// TIA Portal V16 export
// export: Created 2023-03-29T11:04:42.156007Z, ExportSetting WithDefaults, DisplayName Totally Integrated Automation Portal, DisplayVersion V16 Update 6, DisplayName TIA Portal Version Control Interface, DisplayVersion V16 Update 2, DisplayName TIA Portal Openness, DisplayVersion V16 Update 6, DisplayName STEP 7 Professional, DisplayVersion V16 Update 6, DisplayName STEP 7 Safety, DisplayVersion V16, DisplayName WinCC Advanced, DisplayVersion V16 Update 6
DATA_BLOCK "dbMasterData"   // DB35
{ S7_Optimized_Access := 'FALSE' }
VERSION : 0.1
// stored: AutoNumber false, DBAccessibleFromOPCUA true, IsOnlyStoredInLoadMemory false, IsWriteProtectedInAS false
   VAR
      data5_Wielkość_przeływu_Adres_0 { S7_SetPoint := 'True'} : "typeDataMPP04_Int";   // wielkość przepływu / Wartość aktualnego przepływu
      data5_Licznik_objętość_VF_Adres_2 : "typeDataMPP04_Int";   // licznik objętości VF / Stan licznika objętości dla przepływu w przód VF
      data5_Licznik_objętość_VR_Adres_4 { S7_SetPoint := 'True'} : "typeDataMPP04_Int";   // licznik objętości VR / Stan licznika objętości dla przepływu w tył VR
      data5_Licznik_różnicowy_VD_Adres_6 { S7_SetPoint := 'True'} : "typeDataMPP04_Int";   // licznik różnicy / Stan bieżącego różnicowego licznika objętości VD
      data5_Stan_licz_bjętości_GF_Adres_8 { S7_SetPoint := 'True'} : "typeDataMPP04_Int";   // licznik objetosci GF / Stan głównego licznika objętości dla przepływu w przód GF
      data5_Stan_licz_bjętości_GR_Adres_10 { S7_SetPoint := 'True'} : "typeDataMPP04_Int";   // licznik objetości GR / Sta ngłownego licznika objętości dla przepływu w tył GR
      data5_Stan_licz_rózicowego_obj_GD_Adres_12 { S7_SetPoint := 'True'} : "typeDataMPP04_Int";   // licznik róznicowy / Stan głownego licznika różnicowego GD
      data5_Stan_urządzenia_1000 { S7_SetPoint := 'True'} : "typeDataInverter_Word";   // stan urządzenia / 8-przekrodzony zakres pracy przetwornika, 20-otwarty obwód cewki, 21zwarcie w obwodzie cewki, 26-brak cieczy w czujniku
      data6_Wielkość_przeływu_Adres_0 { S7_SetPoint := 'True'} : "typeDataMPP04_Int";   // wielkość przepływu / Wartość aktualnego przepływu
      data6_Licznik_objętość_VF_Adres_2 { S7_SetPoint := 'True'} : "typeDataMPP04_Int";   // licznik objętości VF / Stan licznika objętości dla przepływu w przód VF
      data6_Licznik_objętość_VR_Adres_4 { S7_SetPoint := 'True'} : "typeDataMPP04_Int";   // licznik objętości VR / Stan licznika objętości dla przepływu w tył VR
      data6_Licznik_różnicowy_VD_Adres_6 { S7_SetPoint := 'True'} : "typeDataMPP04_Int";   // licznik różnicy / Stan bieżącego różnicowego licznika objętości VD
      data6_Stan_licz_bjętości_GF_Adres_8 { S7_SetPoint := 'True'} : "typeDataMPP04_Int";   // licznik objetosci GF / Stan głównego licznika objętości dla przepływu w przód GF
      data6_Stan_licz_bjętości_GR_Adres_10 { S7_SetPoint := 'True'} : "typeDataMPP04_Int";   // licznik objetości GR / Sta ngłownego licznika objętości dla przepływu w tył GR
      data6_Stan_licz_rózicowego_obj_GD_Adres_12 { S7_SetPoint := 'True'} : "typeDataMPP04_Int";   // licznik róznicowy / Stan głownego licznika różnicowego GD
      data6_Stan_urządzenia_1000 { S7_SetPoint := 'True'} : "typeDataInverter_Word";   // stan urządzenia / 8-przekrodzony zakres pracy przetwornika, 20-otwarty obwód cewki, 21zwarcie w obwodzie cewki, 26-brak cieczy w czujniku
      data26_Inver_Control_word_416000_Fal { S7_SetPoint := 'True'} : "typeDataInverter_Word";   // Sowo komtrolneCTW falownika [Uint16, index 0]
      data26_Inver_setpoint_ref_416020_Fal { S7_SetPoint := 'True'} : "typeDataInverter_Word";   // Słowo wartość zadana Hz [Int16, index -1]
      data26_Inver_Status_word_416030_Fal { S7_SetPoint := 'True'} : "typeDataInverter_Word";   // Słowo statusu STW falownika [Uint16, index 0]
      data26_Inver_Frequency_416130_Fal { S7_SetPoint := 'True'} : "typeDataInverter_Word";   // Słowo częstotliwość na wyjściu [Uint16, index -1]
      data26_Inver_MotorCurrent_416140_Fal { S7_SetPoint := 'True'} : "typeDataInverter_Word";   // Słowo częstotliwość na wyjściu [Uint16, index -2]
      data26_Inver_DC_Voltage_416300_Fal { S7_SetPoint := 'True'} : "typeDataInverter_Word";   // Słowo napięcia DC na szynie [Uint16, index 0]
      data26_Inver_Temp_416340_Fal { S7_SetPoint := 'True'} : "typeDataInverter_Word";   // Słowo temperatura invertera [Uint8, index 0]
      data26_Inver_NomCurrent_416360_Fal { S7_SetPoint := 'True'} : "typeDataInverter_Word";   // Słowo nominalna wartośc prądu falonika[Uint16, index -2]
      data26_Inver_MaxCurrent_416370_Fal { S7_SetPoint := 'True'} : "typeDataInverter_Word";   // Słowo max prąd falownika [Uint16, index -2]
      data26_Inver_InDigit_416600_Fal { S7_SetPoint := 'True'} : "typeDataInverter_Word";   // Słowo mampa wejść 18,19,27,33 [Uint16, index -0]
      data26_Inver_HourWork_415010_Fal { S7_SetPoint := 'True'} : "typeDataInverter_DWord";   // Podwójne słowo czasu pracy falownika [Int32, index -0]
      data26_Inver_OverTemp_415040_Fal { S7_SetPoint := 'True'} : "typeDataInverter_Word";   // Sowo statusu przekroczenie temperatury[Uint16, index 0]
      data26_Inver_OverVolts_415050_Fal { S7_SetPoint := 'True'} : "typeDataInverter_Word";   // Sowo statusu przekroczenie napięcia[Uint16, index 0]
      data_RTU_value_0 { S7_SetPoint := 'True'} : "typeDataMPP04_real";   // Wartość 0.0 pomocnicza wyświetlana podczas błędu pomiaru
   END_VAR
BEGIN
   data_RTU_value_0.data[0] := 0.0;
END_DATA_BLOCK
